// TIA Portal V20 export
FUNCTION "StringToDTL" : DTL   // FC20225, LAD
{ S7_Optimized_Access := 'TRUE' }
// stored: AutoNumber false, SetENOAutomatically false
   VAR_INPUT
      inString : String;   // Date as String tag
   END_VAR
   VAR_OUTPUT
      error : Bool;   // "0" = no error; "1" = error
      status : Word;   // status and error codes
   END_VAR
   VAR_TEMP
      format : Bool;   // Format of inString/ 0=traditional; 1=international
      tempCounter : Int;   // -
      tempOutput : DTL;   // -
      tempYear : String;   // -
      tempMonth : String;   // -
      tempDay : String;   // -
      tempHour : String;   // -
      tempMinute : String;   // -
      tempSecond : String;   // -
      tempNanosecond : String;   // -
      tempPosYear : USInt;   // -
      tempPosMonth : USInt;   // -
      tempPosDay : USInt;   // -
      tempPosHour : USInt;   // -
      tempPosMinute : USInt;   // -
      tempPosSecond : USInt;   // -
      tempPosNanosecond : USInt;   // -
      tempPosSepYearMonth : USInt;   // -
      tempPosSepMonthDay : USInt;   // -
      tempPosSepHourMinute : USInt;   // -
      tempPosSepMinuteSecond : USInt;   // -
      tempPosSepSecondNanosecond : USInt;   // -
   END_VAR
   VAR CONSTANT
      NO_ERROR : Word := 16#0000;   // -
      NO_CURRENT_JOBS : Word := 16#7000;   // -
      ERROR_FORMAT_YEAR : Word := 16#8201;   // -
      ERROR_FORMAT_MONTH : Word := 16#8202;   // -
      ERROR_FORMAT_DAY : Word := 16#8203;   // -
      ERROR_FORMAT_HOUR : Word := 16#8204;   // -
      ERROR_FORMAT_MINUTE : Word := 16#8205;   // -
      ERROR_FORMAT_SECOND : Word := 16#8206;   // -
      ERROR_FORMAT_NANOSECOND : Word := 16#8207;   // -
      INITIAL_VALUE : DTL := DTL#1970-01-01-00:00:00.0;   // -
   END_VAR
   // Ret_Val : Date as DTL tag
BEGIN

REGION Network 1 (SCL): Set initial parameters
   #error := FALSE;
   #status := #NO_ERROR;

   IF #inString = ''
   THEN
       #StringToDTL := #INITIAL_VALUE;
       #status := #NO_CURRENT_JOBS;
       RETURN;
   END_IF;

   #format := 1;
END_REGION

REGION Network 2 (SCL): Set format parameters for input string
   IF  #format
   THEN
       #tempPosYear := 1;                          // DTL  | Y| Y| Y| Y| -| M| M| -| D| D|  | H| H| :| M| M| :| S| S| .|NS|NS|NS|NS|NS|NS|NS|NS|NS
       #tempPosMonth := 6;                         // -----|--|--|--|--|--|--|--|--|--|--|--|--|--|--|--|--|--|--|--|--|--|--|--|--|--|--|--|--|--
       #tempPosDay := 9;                           // Pos  | 1| 2| 3| 4| 5| 6| 7| 8| 9|10|11|12|13|14|15|16|17|18|19|20|21|22|23|24|25|26|27|28|29
       #tempPosHour := 12;
       #tempPosMinute := 15;
       #tempPosSecond := 18;
       #tempPosNanosecond := 21;
       #tempPosSepYearMonth := 5;
       #tempPosSepMonthDay := 8;
       #tempPosSepHourMinute := 14;
       #tempPosSepMinuteSecond := 17;
       #tempPosSepSecondNanosecond := 20;
   ELSE
       #tempPosYear := 7;                          // DTL  | D| D| -| M| M| -| Y| Y| Y| Y|  | H| H| :| M| M| :| S| S| .|NS|NS|NS|NS|NS|NS|NS|NS|NS
       #tempPosMonth := 4;                         // -----|--|--|--|--|--|--|--|--|--|--|--|--|--|--|--|--|--|--|--|--|--|--|--|--|--|--|--|--|--
       #tempPosDay := 1;                           // Pos  | 1| 2| 3| 4| 5| 6| 7| 8| 9|10|11|12|13|14|15|16|17|18|19|20|21|22|23|24|25|26|27|28|29
       #tempPosHour := 12;
       #tempPosMinute := 15;
       #tempPosSecond := 18;
       #tempPosNanosecond := 21;
       #tempPosSepYearMonth := 6;
       #tempPosSepMonthDay := 3;
       #tempPosSepHourMinute := 14;
       #tempPosSepMinuteSecond := 17;
       #tempPosSepSecondNanosecond := 20;
   END_IF;
END_REGION

REGION Network 3 (SCL): Separating the input string into components of DTL
   #tempYear := MID(IN := #inString, L := 4, P := #tempPosYear);
   #tempMonth := MID(IN := #inString, L := 2, P := #tempPosMonth);
   #tempDay := MID(IN := #inString, L := 2, P := #tempPosDay);
   #tempHour := MID(IN := #inString, L := 2, P := #tempPosHour);
   #tempMinute := MID(IN := #inString, L := 2, P := #tempPosMinute);
   #tempSecond := MID(IN := #inString, L := 2, P := #tempPosSecond);
   #tempNanosecond := MID(IN := #inString, L := 9, P := #tempPosNanosecond);
END_REGION

REGION Network 4 (SCL): Replacing of the "blan" in the nanosecondstring by "0"
   //==> Effect:   xx.1 --> xx.1 AND NOT xx.1 --> xx.000000001
   FOR #tempCounter := 1 TO 9 BY 1
   DO
       IF #tempNanosecond[#tempCounter] = ' '
       THEN
           #tempNanosecond[#tempCounter] := '0';
       END_IF;
   END_FOR;
END_REGION

REGION Network 5 (SCL): Converting separated String components into DTL values
   STRG_VAL(FORMAT := W#16#0000,
            IN := #tempYear,
            OUT => #tempOutput.YEAR,
            P := 1);

   STRG_VAL(FORMAT := W#16#0000,
            IN := #tempMonth,
            OUT => #tempOutput.MONTH,
            P := 1);

   STRG_VAL(FORMAT := W#16#0000,
            IN := #tempDay,
            OUT => #tempOutput.DAY,
            P := 1);

   STRG_VAL(FORMAT := W#16#0000,
            IN := #tempHour,
            OUT => #tempOutput.HOUR,
            P := 1);

   STRG_VAL(FORMAT := W#16#0000,
            IN := #tempMinute,
            OUT => #tempOutput.MINUTE,
            P := 1);

   STRG_VAL(FORMAT := W#16#0000,
            IN := #tempSecond,
            OUT => #tempOutput.SECOND,
            P := 1);

   STRG_VAL(FORMAT := W#16#0000,
            IN := #tempNanosecond,
            OUT => #tempOutput.NANOSECOND,
            P := 1);
END_REGION

REGION Network 6 (SCL): Format check
   IF (#tempOutput.YEAR < 1970) OR (2262 < #tempOutput.YEAR)
   THEN
       #error := TRUE;
       #status := #ERROR_FORMAT_YEAR;
       #StringToDTL := #INITIAL_VALUE;
       RETURN;
   END_IF;

   IF (#tempOutput.MONTH < 1) OR (12 < #tempOutput.MONTH)
   THEN
       #error := TRUE;
       #status := #ERROR_FORMAT_MONTH;
       #StringToDTL := #INITIAL_VALUE;
       RETURN;
   END_IF;

   IF (#tempOutput.DAY < 1) OR (31 < #tempOutput.DAY)
   THEN
       #error := TRUE;
       #status := #ERROR_FORMAT_DAY;
       #StringToDTL := #INITIAL_VALUE;
       RETURN;
   END_IF;

   IF (#tempOutput.HOUR < 0) OR (23 < #tempOutput.HOUR)
   THEN
       #error := TRUE;
       #status := #ERROR_FORMAT_HOUR;
       #StringToDTL := #INITIAL_VALUE;
       RETURN;
   END_IF;

   IF (#tempOutput.MINUTE < 0) OR (59 < #tempOutput.MINUTE)
   THEN
       #error := TRUE;
       #status := #ERROR_FORMAT_MINUTE;
       #StringToDTL := #INITIAL_VALUE;
       RETURN;
   END_IF;

   IF (#tempOutput.SECOND < 0) OR (59 < #tempOutput.SECOND)
   THEN
       #error := TRUE;
       #status := #ERROR_FORMAT_SECOND;
       #StringToDTL := #INITIAL_VALUE;
       RETURN;
   END_IF;

   IF (#tempOutput.NANOSECOND < 0) OR (999999999 < #tempOutput.NANOSECOND)
   THEN
       #error := TRUE;
       #status := #ERROR_FORMAT_NANOSECOND;
       #StringToDTL := #INITIAL_VALUE;
       RETURN;
   END_IF;
END_REGION

REGION Network 7 (SCL): String to DTL
   #StringToDTL := #tempOutput;
END_REGION
END_FUNCTION
